FUNCTION_BLOCK FB_BaseHMIControlElement_Command EXTENDS FB_BaseHMIComponent_Command IMPLEMENTS ITF_BaseHMIControlElement_Command
VAR
END_VAR

END_FUNCTION_BLOCK

(* stored: Version 1.1.0.1
   POU FB_BaseHMIControlElement_Command: Id {e607bb09-e421-057d-2449-fbc2bfa87169}, SpecialFunc None *)
